Yaskawa INFORM job: MT_PRE-PROCESS.JBI

/JOB
//NAME MT_PRE-PROCESS
//POS
///NPOS 0,0,0,2,0,0
///USER 1
///TOOL 0
///POSTYPE USER
///RECTAN
///RCONF 0,0,0,0,0,0,0,0,0,0,0,0,0,0,0,0,0,0,0,0,0,0,0,0
P00052=162.550,-20.884,-140.049,-88.7831,37.5464,-63.7084
P00053=0.000,0.000,50.000,0.0000,0.0000,0.0000
//INST
///DATE 2023/11/21 13:23
///ATTR SC,RW
///GROUP1 RB1
NOP
SET P053 P052
SET I000 0
SET I001 0
SET I002 0
SET B000 1
SET B001 0
END
